TYPE TYP_HW_L4000_EXT_STATUS :
STRUCT
	Acknowledge AT %I* : ARRAY[0..7] OF BOOL;
END_STRUCT
END_TYPE

(* stored: Version 1.1.0.1, ProductVersion 3.1.4024.12
   DUT TYP_HW_L4000_EXT_STATUS: Id {bf07d50a-9e1c-40e9-a169-5ee521d4e453} *)
